# EPICS autosave request: iocStats/iocAdminSoft_settings.req
$(IOC):ACCESS
